INTERFACE ITF_MCHMIPrepareDataForScreenExtension

METHOD PUBLIC LinkExtensionDisplay : BOOL
VAR_INPUT
	fbExtendedDisplay			: ITF_MCHMIDisplayExtension;
END_VAR
END_METHOD

END_INTERFACE

(* stored: Version 1.1.0.1
   Itf ITF_MCHMIPrepareDataForScreenExtension: Id {3eba7dd6-534a-0869-080a-4ac7386c187f}
   Method LinkExtensionDisplay: Id {59992657-2331-01e2-1f12-054db1ae02e6} *)
